FUNCTION_BLOCK FB_FallibleSTRING IMPLEMENTS I_FallibleSTRING
VAR
    bError : BOOL;
    sErrorMsg : T_MaxString;
    sVal : STRING;
END_VAR

METHOD ClearError

bError := FALSE;
sErrorMsg := '';
END_METHOD

METHOD GetError : BOOL

GetError := bError;
END_METHOD

METHOD GetErrorMsg : Tc2_System.T_MaxString

GetErrorMsg := sErrorMsg;
END_METHOD


METHOD SetError
VAR_INPUT
    sMsg	: Tc2_System.T_MaxString;
END_VAR

bError := TRUE;
sErrorMsg := sMsg;
END_METHOD

PROPERTY Val : STRING
GET

Val := sVal;
END_GET
SET

sVal := Val;
END_SET
END_PROPERTY

END_FUNCTION_BLOCK

(* stored: Version 1.1.0.1, ProductVersion 3.1.4022.18
   POU FB_FallibleSTRING: Id {1b890771-a463-46cb-9b7e-1d661e78cbf7}, SpecialFunc None
   Method ClearError: Id {a565d3a2-0dec-45b5-bd57-56476d6a51d4}
   Method GetError: Id {1d1435eb-3c03-49e9-b64b-dc70a252707a}
   Method GetErrorMsg: Id {abc96ace-b996-4094-bf54-60d2eedbbe7c}
   Method SetError: Id {5d0ab8e7-9945-4568-be08-ad0fc810caaf}
   Property Val: Id {aeada6db-8db7-440a-a0bb-2bd912d36b46}
   Get Get: Id {962bb435-90f6-4ca7-931b-3d84dee457c0}
   Set Set: Id {3c84aeb3-1be6-4983-879f-26b7332097e7} *)
